{attribute addProperty BoxType "EJ7031-0000-0026"}
{attribute addProperty Id "StatusAT %I*Status_06A4ECA2162"}
{attribute addProperty CRC "1691957059"}
{attribute addProperty SizeInBites "16"}
{attribute addProperty SizeInBytes "2"}
TYPE STM_Status_64D93743 :
STRUCT
	{attribute addProperty Name "Status"}
	Status AT %I* : Status_06A4ECA2;
END_STRUCT
END_TYPE

(* stored: Version 1.2.0.0, ProductVersion 3.1.4024.9
   DUT STM_Status_64D93743: Id {865a3776-eeeb-4558-bf5a-1849c9a097aa} *)
